// TIA Portal V20 export
ORGANIZATION_BLOCK "Main"   // OB1, LAD, ProgramCycle
TITLE = "Main Program Sweep (Cycle)"
{ S7_Optimized_Access := 'TRUE' }
// stored: SetENOAutomatically false
   VAR_INPUT
      Initial_Call : Bool;   // Initial call of this OB
      Remanence : Bool;   // =True, if remanent data are available
   END_VAR
BEGIN

REGION Network 2: First Cycle
   // Set bit to true in first cycle, and false in all other cycles
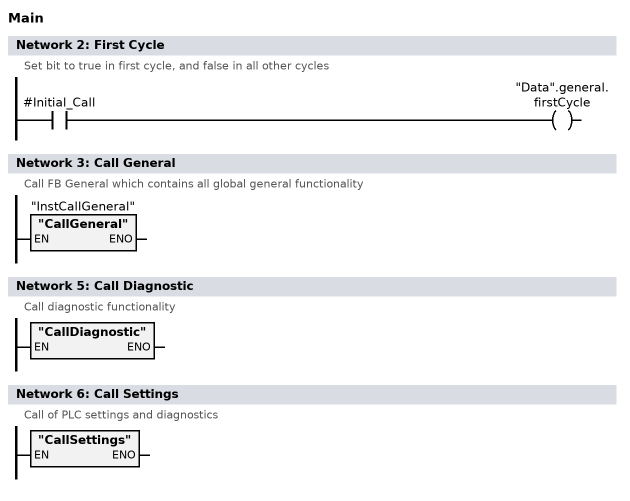
   RUNG wire#powerrail
      Contact( #Initial_Call )
      Coil( "Data".general.firstCycle )
   END_RUNG
   // the same network as SCL:
   "Data".general.firstCycle := #Initial_Call;
END_REGION

REGION Network 3: Call General
   // Call FB General which contains all global general functionality
   RUNG wire#powerrail
      "InstCallGeneral"()
   END_RUNG
   // the same network as SCL:
   "InstCallGeneral"();   // "CallGeneral"
END_REGION

REGION Network 4: Call Manual Operation Lines
   // Not used in Automation Framework Basic
END_REGION

REGION Network 5: Call Diagnostic
   // Call diagnostic functionality
   RUNG wire#powerrail
      "CallDiagnostic"()
   END_RUNG
   // the same network as SCL:
   "CallDiagnostic"();
END_REGION

REGION Network 6: Call Settings
   // Call of PLC settings and diagnostics
   RUNG wire#powerrail
      "CallSettings"()
   END_RUNG
   // the same network as SCL:
   "CallSettings"();
END_REGION
END_ORGANIZATION_BLOCK
